// TIA Portal V17 export
// export: Created 2025-03-07T09:19:16.6359024Z, ExportSetting WithDefaults, DisplayName Totally Integrated Automation Portal, DisplayVersion V17 Update 8, DisplayName TIA Portal Openness, DisplayVersion V17 Update 8, DisplayName TIA Portal Version Control Interface, DisplayVersion V17, DisplayName SINAMICS Startdrive Advanced, DisplayVersion V17 SP2, DisplayName SINAMICS Startdrive G110M, G120, G120C, G120D, G120P, G115D, DisplayVersion V17 SP2, DisplayName SINAMICS Startdrive G130, G150, S120, S150, SINAMICS MV, S210, DisplayVersion V17 SP2, DisplayName STEP 7 Professional, DisplayVersion V17 Update 8, DisplayName SINUMERIK ONE STEP 7 Toolbox, DisplayVersion V17 Update 12, DisplayName SINUMERIK 840D sl STEP 7 Toolbox, DisplayVersion V17 Update 12, DisplayName STEP 7 Safety, DisplayVersion V17 Update 6, DisplayName WinCC Advanced, DisplayVersion V17 Update 8
DATA_BLOCK "DB7231_MAX_OUTPUT_INTERLOCK_GENERAL"   // DB7231
{ S7_Optimized_Access := 'FALSE' }
VERSION : 0.1
// stored: AutoNumber false, DBAccessibleFromOPCUA true, DBAccessibleFromWebserver true, IsOnlyStoredInLoadMemory false, IsWriteProtectedInAS false
   VAR
      STATION_ALARMS : Struct   // STATION ALARMS
         STATION_1_INFEED : Bool;   // STATION 1 INFEED ALARMS
         STATION_2_OUTFEED : Bool;   // STATION 2 OUTFEED ALARMS
         STATION_3_UNIT_01 : Bool;   // STATION 3 UNIT 01 ALARMS
         STATION_4_UNIT_02 : Bool;   // STATION 4 UNIT 02 ALARMS
         STATION_5_COOLING_1 : Bool;   // STATION 5 COOLING 1 ALARMS
         STATION_5_COOLING_2 : Bool;   // STATION 5 COOLING 2 ALARMS
         STATION_5_COOLING_3 : Bool;   // STATION 5 COOLING 3 ALARMS
         STATION_5_COOLING_4 : Bool;   // STATION 5 COOLING 4 ALARMS
         STATION_6_INSPECTION : Bool;   // STATION 6 INSPECTION ALARMS
         STATION_7_MASTER_PART : Bool;   // STATION 7 MASTER PART ALARMS
         STATION_8_QUALITY_AND_REJECT : Bool;   // STATION 8 QUALITY AND REJECT ALARMS
         STATION_9_PART_ROTATION_1 : Bool;   // STATION 9 PART ROTATION 1 ALARMS
         STATION_10_PART_ROTATION_2 : Bool;   // STATION 10 PART ROTATION 2 ALARMS
         STATION_11_PART_ROTATION_3 : Bool;   // STATION 11 PART ROTATION 3 ALARMS
         STATION_21_ROBOT_1 : Bool;   // STATION 21 ROBOT 1 ALARMS
         STATION_22_ROBOT_2 : Bool;   // STATION 22 ROBOT 2 ALARMS
      END_STRUCT;
      STATION_WARNINGS : Struct
         STATION_1_INFEED : Bool;   // STATION 1 INFEED WARNINGS
         STATION_2_OUTFEED : Bool;   // STATION 2 OUTFEED WARNINGS
         STATION_3_UNIT_01 : Bool;   // STATION 3 UNIT 01 WARNINGS
         STATION_4_UNIT_02 : Bool;   // STATION 4 UNIT 02 WARNINGS
         STATION_5_COOLING_1 : Bool;   // STATION 5 COOLING 1 WARNINGS
         STATION_5_COOLING_2 : Bool;   // STATION 5 COOLING 2 WARNINGS
         STATION_5_COOLING_3 : Bool;   // STATION 5 COOLING 3 WARNINGS
         STATION_5_COOLING_4 : Bool;   // STATION 5 COOLING 4 WARNINGS
         STATION_6_INSPECTION : Bool;   // STATION 6 INSPECTION WARNINGS
         STATION_7_MASTER_PART : Bool;   // STATION 7 MASTER PART WARNINGS
         STATION_8_QUALITY_AND_REJECT : Bool;   // STATION 8 QUALITY AND REJECT WARNINGS
         STATION_9_PART_ROTATION_1 : Bool;   // STATION 9 PART ROTATION 1 WARNINGS
         STATION_10_PART_ROTATION_2 : Bool;   // STATION 10 PART ROTATION 2 WARNINGS
         STATION_11_PART_ROTATION_3 : Bool;   // STATION 11 PART ROTATION 3 WARNINGS
         STATION_21_ROBOT_1 : Bool;   // STATION 21 ROBOT 1 WARNINGS
         STATION_22_ROBOT_2 : Bool;   // STATION 22 ROBOT 2 WARNINGS
      END_STRUCT;
      STATION_PART_STATUS : Struct
         STATION_1_INFEED_PART_PRESENT : Bool;   // STATION 1 INFEED PART PRESENT
         STATION_1_INFEED_PART_OK : Bool;   // STATION 1 INFEED PART OK
         STATION_1_INFEED_PART_REJECTED : Bool;   // STATION 1 INFEED PART REJECTED
         STATION_1_INFEED_QUALITY_PART : Bool;   // STATION 1 INFEED QUALITY PART
         STATION_2_OUTFEED_PART_PRESENT : Bool;   // STATION 2 OUTFEED PART PRESENT
         STATION_2_OUTFEED_PART_OK : Bool;   // STATION 2 OUTFEED PART OK
         STATION_2_OUTFEED_PART_REJECTED : Bool;   // STATION 2 OUTFEED PART REJECTED
         STATION_2_OUTFEED_QUALITY_PART : Bool;   // STATION 2 OUTFEED QUALITY PART
         STATION_5_COOLING_1_PART_PRESENT : Bool;   // STATION 5 COOLING 1 PART PRESENT
         STATION_5_COOLING_1_PART_OK : Bool;   // STATION 5 COOLING 1 PART OK
         STATION_5_COOLING_1_PART_REJECTED : Bool;   // STATION 5 COOLING 1 PART REJECTED
         STATION_5_COOLING_1_QUALITY_PART : Bool;   // STATION 5 COOLING 1 QUALITY PART
         STATION_5_COOLING_2_PART_PRESENT : Bool;   // STATION 5 COOLING 2 PART PRESENT
         STATION_5_COOLING_2_PART_OK : Bool;   // STATION 5 COOLING 2 PART OK
         STATION_5_COOLING_2_PART_REJECTED : Bool;   // STATION 5 COOLING 2 PART REJECTED
         STATION_5_COOLING_2_QUALITY_PART : Bool;   // STATION 5 COOLING 2 QUALITY PART
         STATION_5_COOLING_3_PART_PRESENT : Bool;   // STATION 5 COOLING 3 PART PRESENT
         STATION_5_COOLING_3_PART_OK : Bool;   // STATION 5 COOLING 3 PART OK
         STATION_5_COOLING_3_PART_REJECTED : Bool;   // STATION 5 COOLING 3 PART REJECTED
         STATION_5_COOLING_3_QUALITY_PART : Bool;   // STATION 5 COOLING 3 QUALITY PART
         STATION_5_COOLING_4_PART_PRESENT : Bool;   // STATION 5 COOLING 4 PART PRESENT
         STATION_5_COOLING_4_PART_OK : Bool;   // STATION 5 COOLING 4 PART OK
         STATION_5_COOLING_4_PART_REJECTED : Bool;   // STATION 5 COOLING 4 PART REJECTED
         STATION_5_COOLING_4_QUALITY_PART : Bool;   // STATION 5 COOLING 4 QUALITY PART
         STATION_6_INSPECTION_PART_PRESENT : Bool;   // STATION 6 INSPECTION PART PRESENT
         STATION_6_INSPECTION_PART_OK : Bool;   // STATION 6 INSPECTION PART OK
         STATION_6_INSPECTION_PART_REJECTED : Bool;   // STATION 6 INSPECTION PART REJECTED
         STATION_6_INSPECTION_QUALITY_PART : Bool;   // STATION 6 INSPECTION QUALITY PART
         STATION_7_MASTER_PART_PART_PRESENT : Bool;   // STATION 7 MASTER PART PART PRESENT
         STATION_7_MASTER_PART_PART_OK : Bool;   // STATION 7 MASTER PART PART OK
         STATION_7_MASTER_PART_PART_REJECTED : Bool;   // STATION 7 MASTER PART PART REJECTED
         STATION_7_MASTER_PART_QUALITY_PART : Bool;   // STATION 7 MASTER PART QUALITY PART
         STATION_8_QUALITY_AND_REJECT_PART_PRESENT : Bool;   // STATION 8 QUALITY AND REJECT PART PRESENT
         STATION_8_QUALITY_AND_REJECT_PART_OK : Bool;   // STATION 8 QUALITY AND REJECT PART OK
         STATION_8_QUALITY_AND_REJECT_PART_REJECTED : Bool;   // STATION 8 QUALITY AND REJECT PART REJECTED
         STATION_8_QUALITY_AND_REJECT_QUALITY_PART : Bool;   // STATION 8 QUALITY AND REJECT QUALITY PART
         STATION_9_PART_ROTATION_1_PART_PRESENT : Bool;   // STATION 9 PART ROTATION 1 PART PRESENT
         STATION_9_PART_ROTATION_1_PART_OK : Bool;   // STATION 9 PART ROTATION 1 PART OK
         STATION_9_PART_ROTATION_1_PART_REJECTED : Bool;   // STATION 9 PART ROTATION 1 PART REJECTED
         STATION_9_PART_ROTATION_1_QUALITY_PART : Bool;   // STATION 9 PART ROTATION 1 QUALITY PART
         STATION_10_PART_ROTATION_2_PART_PRESENT : Bool;   // STATION 10 PART ROTATION 2 PART PRESENT
         STATION_10_PART_ROTATION_2_PART_OK : Bool;   // STATION 10 PART ROTATION 2 PART OK
         STATION_10_PART_ROTATION_2_PART_REJECTED : Bool;   // STATION 10 PART ROTATION 2 PART REJECTED
         STATION_10_PART_ROTATION_2_QUALITY_PART : Bool;   // STATION 10 PART ROTATION 2 QUALITY PART
         STATION_11_PART_ROTATION_3_PART_PRESENT : Bool;   // STATION 11 PART ROTATION 3 PART PRESENT
         STATION_11_PART_ROTATION_3_PART_OK : Bool;   // STATION 11 PART ROTATION 3 PART OK
         STATION_11_PART_ROTATION_3_PART_REJECTED : Bool;   // STATION 11 PART ROTATION 3 PART REJECTED
         STATION_11_PART_ROTATION_3_QUALITY_PART : Bool;   // STATION 11 PART ROTATION 3 QUALITY PART
         STATION_21_ROBOT_1_PART_PRESENT : Bool;   // STATION 21 ROBOT 1 PART PRESENT
         STATION_21_ROBOT_1_PART_OK : Bool;   // STATION 21 ROBOT 1 PART OK
         STATION_21_ROBOT_1_PART_REJECTED : Bool;   // STATION 21 ROBOT 1 PART REJECTED
         STATION_21_ROBOT_1_QUALITY_PART : Bool;   // STATION 21 ROBOT 1 QUALITY PART
         STATION_22_ROBOT_2_PART_PRESENT : Bool;   // STATION 22 ROBOT 2 PART PRESENT
         STATION_22_ROBOT_2_PART_OK : Bool;   // STATION 22 ROBOT 2 PART OK
         STATION_22_ROBOT_2_PART_REJECTED : Bool;   // STATION 22 ROBOT 2 PART REJECTED
         STATION_22_ROBOT_2_QUALITY_PART : Bool;   // STATION 22 ROBOT 2 QUALITY PART
      END_STRUCT;
      STATION_PART_CELL_STATUS_COLOR : Struct
         STATION_1_INFEED : Int;   // STATION 1 INFEED CELL STATUS COLOR
         STATION_2_OUTFEED : Int;   // STATION 2 OUTFEED CELL STATUS COLOR
         STATION_3_UNIT_01 : Int;   // STATION 3 UNIT 01 CELL STATUS COLOR
         STATION_4_UNIT_02 : Int;   // STATION 4 UNIT 02 CELL STATUS COLOR
         STATION_5_COOLING_1 : Int;   // STATION 5 COOLING 1 CELL STATUS COLOR
         STATION_5_COOLING_2 : Int;   // STATION 5 COOLING 2 CELL STATUS COLOR
         STATION_5_COOLING_3 : Int;   // STATION 5 COOLING 3 CELL STATUS COLOR
         STATION_5_COOLING_4 : Int;   // STATION 5 COOLING 4 CELL STATUS COLOR
         STATION_6_INSPECTION : Int;   // STATION 6 INSPECTION CELL STATUS COLOR
         STATION_7_MASTER_PART : Int;   // STATION 7 MASTER PART CELL STATUS COLOR
         STATION_8_QUALITY_AND_REJECT : Int;   // STATION 8 QUALITY AND REJECT CELL STATUS COLOR
         STATION_9_PART_ROTATION_1 : Int;   // STATION 9 PART ROTATION 1 CELL STATUS COLOR
         STATION_10_PART_ROTATION_2 : Int;   // STATION 10 PART ROTATION 2 CELL STATUS COLOR
         STATION_11_PART_ROTATION_3 : Int;   // STATION 11 PART ROTATION 3 CELL STATUS COLOR
         STATION_21_ROBOT_1 : Int;   // STATION 21 ROBOT 1 CELL STATUS COLOR
         STATION_22_ROBOT_2 : Int;   // STATION 22 ROBOT 2 CELL STATUS COLOR
      END_STRUCT;
      STATION_PART_ID : Struct
         STATION_1_INFEED : Array[0..41] of Char;   // STATION 1 INFEED PART ID
         STATION_2_OUTFEED : Array[0..41] of Char;   // STATION 2 OUTFEED PART ID
         STATION_5_COOLING_1 : Array[0..41] of Char;   // STATION 5 COOLING 1 PART ID
         STATION_5_COOLING_2 : Array[0..41] of Char;   // STATION 5 COOLING 2 PART ID
         STATION_5_COOLING_3 : Array[0..41] of Char;   // STATION 5 COOLING 3 PART ID
         STATION_5_COOLING_4 : Array[0..41] of Char;   // STATION 5 COOLING 4 PART ID
         STATION_6_INSPECTION : Array[0..41] of Char;   // STATION 6 INSPECTION PART ID
         STATION_7_MASTER_PART : Array[0..41] of Char;   // STATION 7 MASTER PART PART ID
         STATION_8_QUALITY_AND_REJECT : Array[0..41] of Char;   // STATION 8 QUALITY AND REJECT PART ID
         STATION_9_PART_ROTATION_1 : Array[0..41] of Char;   // STATION 9 PART ROTATION 1 PART ID
         STATION_10_PART_ROTATION_2 : Array[0..41] of Char;   // STATION 10 PART ROTATION 2 PART ID
         STATION_11_PART_ROTATION_3 : Array[0..41] of Char;   // STATION 11 PART ROTATION 3 PART ID
         STATION_21_ROBOT_1 : Array[0..41] of Char;   // STATION 21 ROBOT 1 PART ID
         STATION_22_ROBOT_2 : Array[0..41] of Char;   // STATION 22 ROBOT 2 PART ID
      END_STRUCT;
      STATION_PART_TYPE : Struct
         STATION_1_INFEED : Byte;   // STATION 1 INFEED PART TYPE
         STATION_2_OUTFEED : Byte;   // STATION 2 OUTFEED PART TYPE
         STATION_5_COOLING_1 : Byte;   // STATION 5 COOLING 1 PART TYPE
         STATION_5_COOLING_2 : Byte;   // STATION 5 COOLING 2 PART TYPE
         STATION_5_COOLING_3 : Byte;   // STATION 5 COOLING 3 PART TYPE
         STATION_5_COOLING_4 : Byte;   // STATION 5 COOLING 4 PART TYPE
         STATION_6_INSPECTION : Byte;   // STATION 6 INSPECTION PART TYPE
         STATION_7_MASTER_PART : Byte;   // STATION 7 MASTER PART PART TYPE
         STATION_8_QUALITY_AND_REJECT : Byte;   // STATION 8 QUALITY AND REJECT PART TYPE
         STATION_9_PART_ROTATION_1 : Byte;   // STATION 9 PART ROTATION 1 PART TYPE
         STATION_10_PART_ROTATION_2 : Byte;   // STATION 10 PART ROTATION 2 PART TYPE
         STATION_11_PART_ROTATION_3 : Byte;   // STATION 11 PART ROTATION 3 PART TYPE
         STATION_21_ROBOT_1 : Byte;   // STATION 21 ROBOT 1 PART TYPE
         STATION_22_ROBOT_2 : Byte;   // STATION 22 ROBOT 2 PART TYPE
      END_STRUCT;
   END_VAR
BEGIN
END_DATA_BLOCK
